PROGRAM PRG_10_CrossCutPosition
VAR
	iStepCrossCut: INT;
//	R_TRIG_CrossCutPosition: R_TRIG;
//	SR_CrossCutPosition: SR;
END_VAR

// bAnyServoError

	IF		NOT bSafetyOK OR IN_FaultReset OR bAutoCrossCut OR bMachineHoming	//OR NOT SR_CrossCutPosition.Q1
	THEN	iStepCrossCut	:=	0;
			bCrossCutPosition := FALSE;
	END_IF
	
(*			R_TRIG_CrossCutPosition(CLK:= bCrossCutPositionEnable AND NOT bMachineHoming AND NOT bAutoCrossCut AND NOT OUT_bSawOn,
									Q=> );	
			SR_CrossCutPosition(SET1:= R_TRIG_CrossCutPosition.Q AND NOT SR_CrossCutPosition.Q1,
								RESET:= (R_TRIG_CrossCutPosition.Q AND SR_CrossCutPosition.Q1) OR NOT bSafetyOK OR IN_FaultReset, 
								Q1=> );		*)
(* HMI Indicators *)
IF bCrossCutPosition THEN
	bCrossCutPositionInProgress := TRUE ;
ELSE
	bCrossCutPositionInProgress := FALSE ;
END_IF

IF NOT bCrossCutPosition
	AND bSawUpLimit
	AND bCarriageCentreRef
	AND bTurretMedianRange
	AND ((lCrossCutEncoderValue > ((lRailLimitLeft + lRailLimitRight)/2) - 40) AND (lCrossCutEncoderValue < ((lRailLimitLeft + lRailLimitRight)/2) + 40))
THEN bCrossCutPositionInPosition := TRUE ;
ELSE bCrossCutPositionInPosition := FALSE ;
END_IF

CASE iStepCrossCut OF
	0:	// Init step
		bTurretCuttingPosCW		:= FALSE; 
		bTurretCuttingPosCCW	:= FALSE;
	    bCarriageCuttingPosLH	:= FALSE;
	    bCarriageCuttingPosRH	:= FALSE;
	    bCrossCutCuttingPosLH	:= FALSE;
	    bCrossCutCuttingPosRH	:= FALSE;
		bZAxisCuttingPos 		:= FALSE;
	
		IF 	IN_bAutoCycleStart		//R_TRIG_CrossCutPosition.Q 
			AND bCrossCutPositionEnable
			AND bSafetyOK 
			AND NOT OUT_bSawOn 
			AND NOT bAutoCrossCut
			AND NOT bMachineHoming
		THEN
			bCrossCutPosition := TRUE ;
			iStepCrossCut := 10 ;
		ELSE
			bCrossCutPosition := FALSE ;
		END_IF
		
	10:	// Raise Z-axis all the way up
	
		IF NOT bSawUpLimit AND bSafetyOK AND bCrossCutPosition THEN
			bZAxisCuttingPos := TRUE ;
		ELSE
			bZAxisCuttingPos := FALSE ; 
			iStepCrossCut := 20 ;
		END_IF
		
	20:	// Move crosscut motor to centre
	 
		IF lCrossCutEncoderValue < ((lRailLimitLeft + lRailLimitRight)/2) - 20 AND bSafetyOK AND bCrossCutPosition THEN
			bCrossCutCuttingPosLH := TRUE ;
			bCrossCutCuttingPosRH := FALSE ;
		ELSIF lCrossCutEncoderValue > ((lRailLimitLeft + lRailLimitRight)/2) + 20 AND bSafetyOK AND bCrossCutPosition THEN
			bCrossCutCuttingPosRH := TRUE ;
			bCrossCutCuttingPosLH := FALSE ;
		ELSIF (lCrossCutEncoderValue > ((lRailLimitLeft + lRailLimitRight)/2) - 20) OR (lCrossCutEncoderValue < ((lRailLimitLeft + lRailLimitRight)/2) + 20) AND bSafetyOK AND bCrossCutPosition THEN
			bCrossCutCuttingPosLH := FALSE ;
			bCrossCutCuttingPosRH := FALSE ;
			iStepCrossCut := 30 ;
		END_IF
	
	30: // Move Carriage to centre	
	
		IF NOT bCarriageCentreRef AND AnalogIn_LREAL_Carriage.Out.rScaled > 20.48 AND bCrossCutPosition AND bSafetyOK THEN
			bCarriageCuttingPosLH := TRUE ;
			bCarriageCuttingPosRH := FALSE ;
		ELSIF NOT bCarriageCentreRef AND AnalogIn_LREAL_Carriage.Out.rScaled < 20.52 AND bCrossCutPosition AND bSafetyOK THEN
			bCarriageCuttingPosRH := TRUE ;
			bCarriageCuttingPosLH := FALSE ;
		ELSIF bCarriageCentreRef AND bCrossCutPosition AND bSafetyOK THEN
			bCarriageCuttingPosRH := FALSE ;
			bCarriageCuttingPosLH := FALSE ;
			iStepCrossCut := 40 ;
		END_IF

	40:	// Rotate turret to Centre
	
		IF NOT bTurretMedianRange AND GVL.Turret_Axis.AchsIn.IstPos > lTurretMedian AND bSafetyOK AND bCrossCutPosition THEN
			bTurretCuttingPosCCW := TRUE ;
			bTurretCuttingPosCW := FALSE ;
		ELSIF NOT bTurretMedianRange AND GVL.Turret_Axis.AchsIn.IstPos < lTurretMedian AND bSafetyOK AND bCrossCutPosition THEN
			bTurretCuttingPosCW := TRUE ;
			bTurretCuttingPosCCW := FALSE ;
		ELSIF bTurretMedianRange AND bSafetyOK AND bCrossCutPosition THEN
			bTurretCuttingPosCW := FALSE ;
			bTurretCuttingPosCCW := FALSE ;
			iStepCrossCut := 0 ;
		END_IF
	

	
(*	50: //Crosscut offset towards the control panel (CUT direction)		// 55.5 < CrosscutHome < 55.75
	
		IF (AnalogIn_LREAL_CrossCut.Out.rScaled < 7) AND bCrossCutPosition AND bSafetyOK THEN
			bCrossCutCuttingPosLH := TRUE ;
			bCrossCutCuttingPosRH := FALSE ;
		ELSIF (AnalogIn_LREAL_CrossCut.Out.rScaled > 8) AND bCrossCutPosition AND bSafetyOK THEN
			bCrossCutCuttingPosRH := TRUE ;
			bCrossCutCuttingPosLH := FALSE ;
		ELSIF (AnalogIn_LREAL_CrossCut.Out.rScaled > 7) AND (AnalogIn_LREAL_CrossCut.Out.rScaled < 8) THEN
			bCrossCutCuttingPosLH := FALSE ;
			bCrossCutCuttingPosRH := FALSE ;
			iStepCrossCut := 0 ;
		END_IF
*)		
END_CASE

END_PROGRAM

(* stored: Version 1.1.0.1, ProductVersion 3.1.4024.15
   POU PRG_10_CrossCutPosition: Id {01508e5e-1a94-4304-b7d0-0ea935e17fc2}, SpecialFunc None *)
